Staubli VAL3: JointTrajPt.dtx

public num nSeq
public num nJoints[10]
public num nVelocity
public num nDuration
